SUBAPPLICATION SClient (* Subapplication Type *)
  (* Standard: 61499-2 *)
  (* Version 1.0, 2019-07-03, dorofeev *)
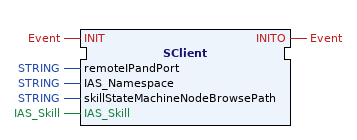
  EVENT_INPUT
    INIT; (* Initialization Request *)
  END_EVENT
  EVENT_OUTPUT
    INITO; (* Initialization Confirm *)
  END_EVENT
  VAR_INPUT
    remoteIPandPort : STRING; (* Input event qualifier *)
    IAS_Namespace : STRING;
    skillStateMachineNodeBrowsePath : STRING;
  END_VAR
  SOCKETS
    IAS_Skill : IAS_Skill;
  END_SOCKETS
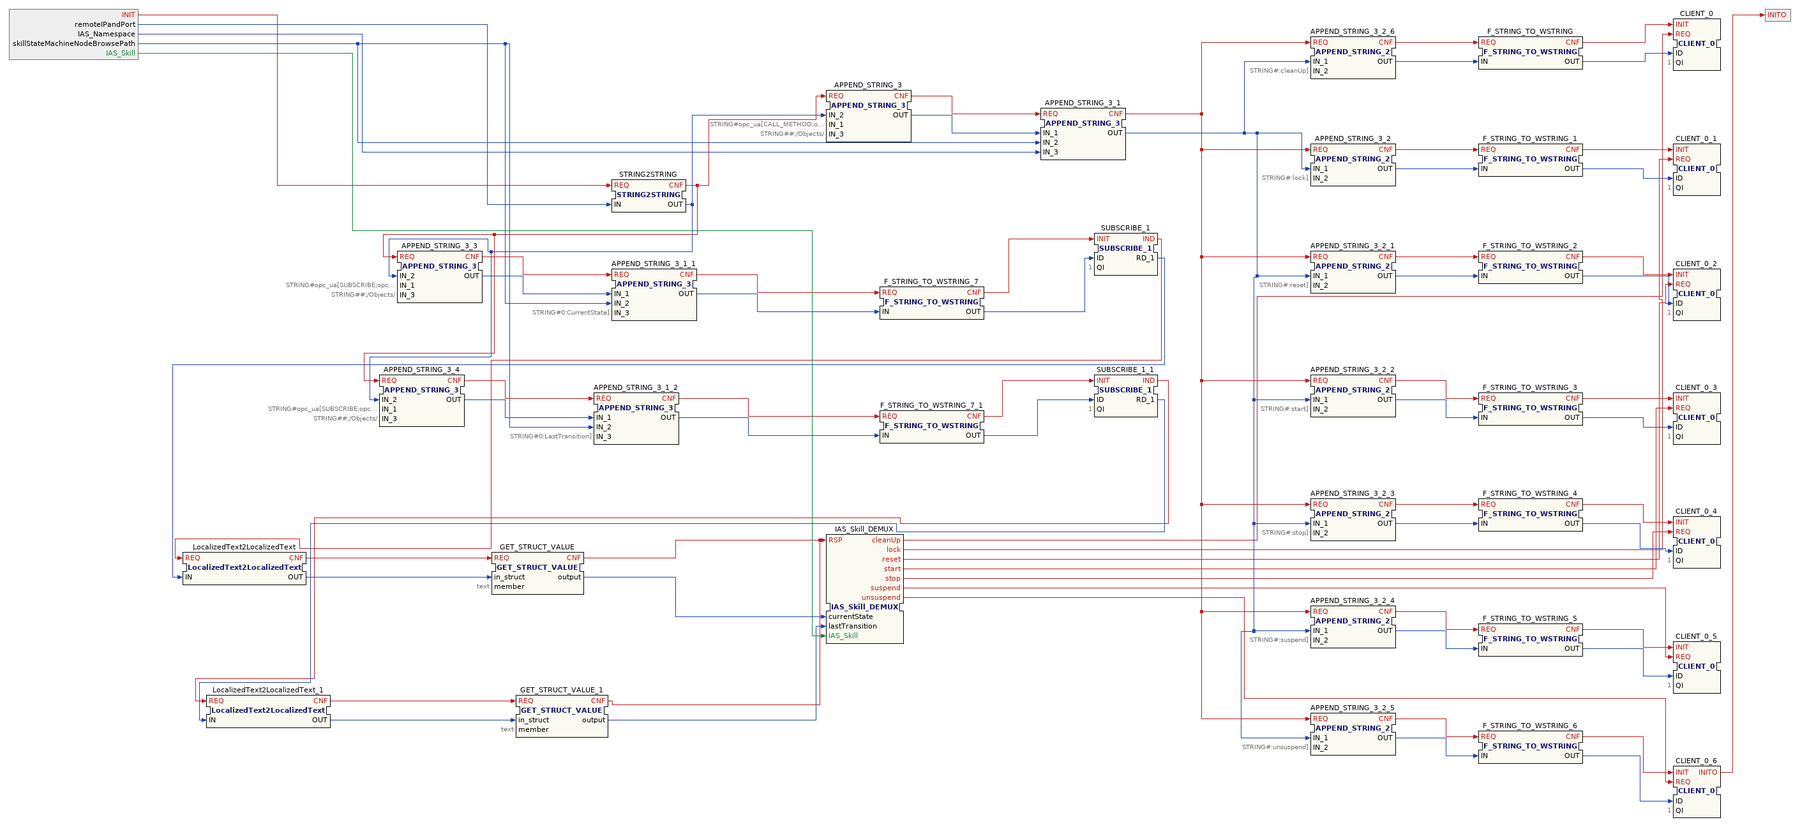
  FBS
    APPEND_STRING_3 : APPEND_STRING_3(IN_1 := STRING#opc_ua[CALL_METHOD;opc.tcp://, IN_3 := STRING##;/Objects/);
    APPEND_STRING_3_1 : APPEND_STRING_3;
    APPEND_STRING_3_2 : APPEND_STRING_2(IN_2 := STRING#:lock]);
    APPEND_STRING_3_2_1 : APPEND_STRING_2(IN_2 := STRING#:reset]);
    APPEND_STRING_3_2_2 : APPEND_STRING_2(IN_2 := STRING#:start]);
    APPEND_STRING_3_2_3 : APPEND_STRING_2(IN_2 := STRING#:stop]);
    APPEND_STRING_3_2_4 : APPEND_STRING_2(IN_2 := STRING#:suspend]);
    APPEND_STRING_3_2_5 : APPEND_STRING_2(IN_2 := STRING#:unsuspend]);
    APPEND_STRING_3_2_6 : APPEND_STRING_2(IN_2 := STRING#:cleanUp]);
    CLIENT_0 : CLIENT_0(QI := 1);
    CLIENT_0_1 : CLIENT_0(QI := 1);
    CLIENT_0_2 : CLIENT_0(QI := 1);
    CLIENT_0_3 : CLIENT_0(QI := 1);
    CLIENT_0_4 : CLIENT_0(QI := 1);
    CLIENT_0_5 : CLIENT_0(QI := 1);
    CLIENT_0_6 : CLIENT_0(QI := 1);
    F_STRING_TO_WSTRING : F_STRING_TO_WSTRING;
    F_STRING_TO_WSTRING_1 : F_STRING_TO_WSTRING;
    F_STRING_TO_WSTRING_2 : F_STRING_TO_WSTRING;
    F_STRING_TO_WSTRING_3 : F_STRING_TO_WSTRING;
    F_STRING_TO_WSTRING_4 : F_STRING_TO_WSTRING;
    F_STRING_TO_WSTRING_5 : F_STRING_TO_WSTRING;
    F_STRING_TO_WSTRING_6 : F_STRING_TO_WSTRING;
    SUBSCRIBE_1 : SUBSCRIBE_1(QI := 1);
    SUBSCRIBE_1_1 : SUBSCRIBE_1(QI := 1);
    APPEND_STRING_3_3 : APPEND_STRING_3(IN_1 := STRING#opc_ua[SUBSCRIBE;opc.tcp://, IN_3 := STRING##;/Objects/);
    APPEND_STRING_3_1_1 : APPEND_STRING_3(IN_3 := STRING#0:CurrentState]);
    APPEND_STRING_3_4 : APPEND_STRING_3(IN_1 := STRING#opc_ua[SUBSCRIBE;opc.tcp://, IN_3 := STRING##;/Objects/);
    APPEND_STRING_3_1_2 : APPEND_STRING_3(IN_3 := STRING#0:LastTransition]);
    F_STRING_TO_WSTRING_7 : F_STRING_TO_WSTRING;
    F_STRING_TO_WSTRING_7_1 : F_STRING_TO_WSTRING;
    STRING2STRING : STRING2STRING;
    IAS_Skill_DEMUX : IAS_Skill_DEMUX;
    GET_STRUCT_VALUE : GET_STRUCT_VALUE(member := text);
    GET_STRUCT_VALUE_1 : GET_STRUCT_VALUE(member := text);
    LocalizedText2LocalizedText_1 : LocalizedText2LocalizedText;
    LocalizedText2LocalizedText : LocalizedText2LocalizedText;
  END_FBS
  EVENT_CONNECTIONS
    APPEND_STRING_3.CNF TO APPEND_STRING_3_1.REQ;
    APPEND_STRING_3_1.CNF TO APPEND_STRING_3_2_6.REQ;
    APPEND_STRING_3_1.CNF TO APPEND_STRING_3_2.REQ;
    APPEND_STRING_3_1.CNF TO APPEND_STRING_3_2_1.REQ;
    APPEND_STRING_3_1.CNF TO APPEND_STRING_3_2_2.REQ;
    APPEND_STRING_3_1.CNF TO APPEND_STRING_3_2_3.REQ;
    APPEND_STRING_3_1.CNF TO APPEND_STRING_3_2_4.REQ;
    APPEND_STRING_3_1.CNF TO APPEND_STRING_3_2_5.REQ;
    APPEND_STRING_3_2_6.CNF TO F_STRING_TO_WSTRING.REQ;
    F_STRING_TO_WSTRING.CNF TO CLIENT_0.INIT;
    APPEND_STRING_3_2.CNF TO F_STRING_TO_WSTRING_1.REQ;
    F_STRING_TO_WSTRING_1.CNF TO CLIENT_0_1.INIT;
    APPEND_STRING_3_2_1.CNF TO F_STRING_TO_WSTRING_2.REQ;
    F_STRING_TO_WSTRING_2.CNF TO CLIENT_0_2.INIT;
    APPEND_STRING_3_2_2.CNF TO F_STRING_TO_WSTRING_3.REQ;
    F_STRING_TO_WSTRING_3.CNF TO CLIENT_0_3.INIT;
    APPEND_STRING_3_2_3.CNF TO F_STRING_TO_WSTRING_4.REQ;
    F_STRING_TO_WSTRING_4.CNF TO CLIENT_0_4.INIT;
    APPEND_STRING_3_2_4.CNF TO F_STRING_TO_WSTRING_5.REQ;
    F_STRING_TO_WSTRING_5.CNF TO CLIENT_0_5.INIT;
    APPEND_STRING_3_2_5.CNF TO F_STRING_TO_WSTRING_6.REQ;
    F_STRING_TO_WSTRING_6.CNF TO CLIENT_0_6.INIT;
    CLIENT_0_6.INITO TO INITO;
    APPEND_STRING_3_3.CNF TO APPEND_STRING_3_1_1.REQ;
    APPEND_STRING_3_4.CNF TO APPEND_STRING_3_1_2.REQ;
    F_STRING_TO_WSTRING_7.CNF TO SUBSCRIBE_1.INIT;
    APPEND_STRING_3_1_1.CNF TO F_STRING_TO_WSTRING_7.REQ;
    APPEND_STRING_3_1_2.CNF TO F_STRING_TO_WSTRING_7_1.REQ;
    F_STRING_TO_WSTRING_7_1.CNF TO SUBSCRIBE_1_1.INIT;
    INIT TO STRING2STRING.REQ;
    STRING2STRING.CNF TO APPEND_STRING_3.REQ;
    STRING2STRING.CNF TO APPEND_STRING_3_3.REQ;
    STRING2STRING.CNF TO APPEND_STRING_3_4.REQ;
    IAS_Skill_DEMUX.cleanUp TO CLIENT_0.REQ;
    IAS_Skill_DEMUX.lock TO CLIENT_0_1.REQ;
    IAS_Skill_DEMUX.reset TO CLIENT_0_2.REQ;
    IAS_Skill_DEMUX.start TO CLIENT_0_3.REQ;
    IAS_Skill_DEMUX.stop TO CLIENT_0_4.REQ;
    IAS_Skill_DEMUX.suspend TO CLIENT_0_5.REQ;
    IAS_Skill_DEMUX.unsuspend TO CLIENT_0_6.REQ;
    LocalizedText2LocalizedText_1.CNF TO GET_STRUCT_VALUE_1.REQ;
    LocalizedText2LocalizedText.CNF TO GET_STRUCT_VALUE.REQ;
    SUBSCRIBE_1_1.IND TO LocalizedText2LocalizedText_1.REQ;
    SUBSCRIBE_1.IND TO LocalizedText2LocalizedText.REQ;
    GET_STRUCT_VALUE.CNF TO IAS_Skill_DEMUX.RSP;
    GET_STRUCT_VALUE_1.CNF TO IAS_Skill_DEMUX.RSP;
  END_CONNECTIONS
  DATA_CONNECTIONS
    APPEND_STRING_3.OUT TO APPEND_STRING_3_1.IN_1;
    skillStateMachineNodeBrowsePath TO APPEND_STRING_3_1.IN_2;
    IAS_Namespace TO APPEND_STRING_3_1.IN_3;
    APPEND_STRING_3_1.OUT TO APPEND_STRING_3_2_6.IN_1;
    APPEND_STRING_3_1.OUT TO APPEND_STRING_3_2.IN_1;
    APPEND_STRING_3_1.OUT TO APPEND_STRING_3_2_1.IN_1;
    APPEND_STRING_3_1.OUT TO APPEND_STRING_3_2_2.IN_1;
    APPEND_STRING_3_1.OUT TO APPEND_STRING_3_2_3.IN_1;
    APPEND_STRING_3_1.OUT TO APPEND_STRING_3_2_4.IN_1;
    APPEND_STRING_3_1.OUT TO APPEND_STRING_3_2_5.IN_1;
    APPEND_STRING_3_2_6.OUT TO F_STRING_TO_WSTRING.IN;
    F_STRING_TO_WSTRING.OUT TO CLIENT_0.ID;
    APPEND_STRING_3_2.OUT TO F_STRING_TO_WSTRING_1.IN;
    F_STRING_TO_WSTRING_1.OUT TO CLIENT_0_1.ID;
    APPEND_STRING_3_2_1.OUT TO F_STRING_TO_WSTRING_2.IN;
    F_STRING_TO_WSTRING_2.OUT TO CLIENT_0_2.ID;
    APPEND_STRING_3_2_2.OUT TO F_STRING_TO_WSTRING_3.IN;
    F_STRING_TO_WSTRING_3.OUT TO CLIENT_0_3.ID;
    APPEND_STRING_3_2_3.OUT TO F_STRING_TO_WSTRING_4.IN;
    F_STRING_TO_WSTRING_4.OUT TO CLIENT_0_4.ID;
    APPEND_STRING_3_2_4.OUT TO F_STRING_TO_WSTRING_5.IN;
    F_STRING_TO_WSTRING_5.OUT TO CLIENT_0_5.ID;
    APPEND_STRING_3_2_5.OUT TO F_STRING_TO_WSTRING_6.IN;
    F_STRING_TO_WSTRING_6.OUT TO CLIENT_0_6.ID;
    APPEND_STRING_3_3.OUT TO APPEND_STRING_3_1_1.IN_1;
    APPEND_STRING_3_4.OUT TO APPEND_STRING_3_1_2.IN_1;
    F_STRING_TO_WSTRING_7.OUT TO SUBSCRIBE_1.ID;
    APPEND_STRING_3_1_1.OUT TO F_STRING_TO_WSTRING_7.IN;
    APPEND_STRING_3_1_2.OUT TO F_STRING_TO_WSTRING_7_1.IN;
    F_STRING_TO_WSTRING_7_1.OUT TO SUBSCRIBE_1_1.ID;
    remoteIPandPort TO STRING2STRING.IN;
    STRING2STRING.OUT TO APPEND_STRING_3.IN_2;
    STRING2STRING.OUT TO APPEND_STRING_3_3.IN_2;
    STRING2STRING.OUT TO APPEND_STRING_3_4.IN_2;
    skillStateMachineNodeBrowsePath TO APPEND_STRING_3_1_1.IN_2;
    skillStateMachineNodeBrowsePath TO APPEND_STRING_3_1_2.IN_2;
    LocalizedText2LocalizedText.OUT TO GET_STRUCT_VALUE.in_struct;
    LocalizedText2LocalizedText_1.OUT TO GET_STRUCT_VALUE_1.in_struct;
    SUBSCRIBE_1_1.RD_1 TO LocalizedText2LocalizedText_1.IN;
    SUBSCRIBE_1.RD_1 TO LocalizedText2LocalizedText.IN;
    GET_STRUCT_VALUE.output TO IAS_Skill_DEMUX.currentState;
    GET_STRUCT_VALUE_1.output TO IAS_Skill_DEMUX.lastTransition;
  END_CONNECTIONS
  ADAPTER_CONNECTIONS
    IAS_Skill TO IAS_Skill_DEMUX.IAS_Skill;
  END_CONNECTIONS
END_SUBAPPLICATION
